Yaskawa INFORM job: MT_CLOSE-DOOR.JBI

/JOB
//NAME MT_CLOSE-DOOR
//POS
///NPOS 0,0,0,0,0,0
//INST
///DATE 2023/11/21 14:28
///ATTR SC,RW
///GROUP1 RB1
NOP
DOUT OT#(531) ON
TIMER T=0.500
DOUT OT#(531) OFF
WAIT IN#(531)=ON
END
